// Mitsubishi GX Works2 project: AJ_woot_drite_test   PLC: FX3U/FX3UC

PROGRAM MAIN
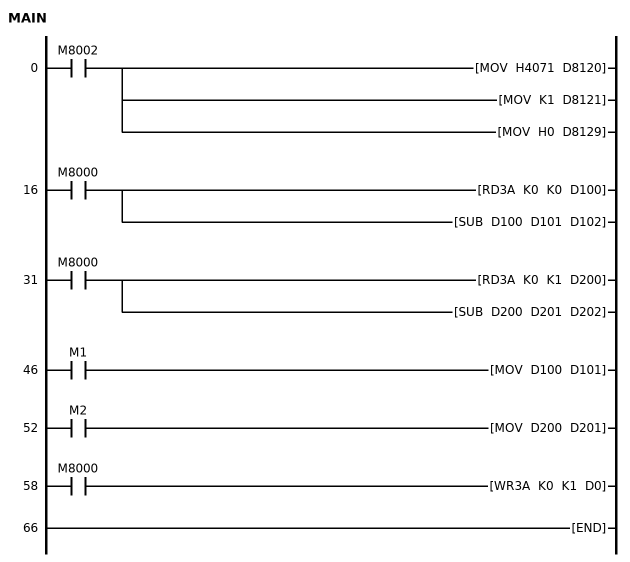
0     LD      M8002
      MOV     H4071 D8120
      MOV     K1 D8121
      MOV     H0 D8129
16    LD      M8000
      RD3A    K0 K0 D100
      SUB     D100 D101 D102
31    LD      M8000
      RD3A    K0 K1 D200
      SUB     D200 D201 D202
46    LD      M1
      MOV     D100 D101
52    LD      M2
      MOV     D200 D201
58    LD      M8000
      WR3A    K0 K1 D0
66    END
END_PROGRAM
